FUNCTION "LAnyAxis_UnpubStatusWordSpeedAxis" : DWord
{ S7_Optimized_Access := 'TRUE' }
AUTHOR : 'tech.team.motioncontrol@siemens.com'
FAMILY : AnyAxis
VERSION : 1.0
   VAR_INPUT
      axis {InstructionName := 'TO_SpeedAxis'; LibVersion := '5.0'} : TO_SpeedAxis;
   END_VAR


BEGIN
	// Read axis parameter
	#LAnyAxis_UnpubStatusWordSpeedAxis := #axis.StatusWord;
END_FUNCTION

